TYPE (* IEC61131-3, Table 14#5 *)
  (* Standard: 1131-3 *)
  (* Version 0.0, 1/8/2024, Cheyan, Schneider Electric, Template *)
  PACKAGE Main;
  {SET_ATTRIBUTE(nxtDataType, z/yCPi5cyPAK7oqqmmhk81uxb23cXjysLjNLfoHyTL1zEyt8VrdsSQhGbSKe8NBJCTf08T6ksxmjxnOgL3ICxEIXf/Atxz/dcJ0RWHyXwP09L80WSH7X0nAlvWsfM5JYDpVl83k9u6YHoILb8OYKAg==)}
  INS_STATUS : STRUCT
    stVal : DINT;
    q : Quality;
    t : TimeStamp;
  END_STRUCT;
END_TYPE
